FUNCTION_BLOCK FB_Homing_Base EXTENDS FB_CyclicFB IMPLEMENTS I_HomingStrategy
VAR
    _Axis     : SPT_Motion_Control.I_BasicAxis;
    _bBusy    : BOOL;
    _bDone    : BOOL;
    _bError   : BOOL;
    _bErrorID : UDINT;
    nStep     : INT;
END_VAR

METHOD Abort
VAR_INPUT
END_VAR
_bBusy := FALSE;
nStep := 0;
END_METHOD

PROPERTY Axis : SPT_Motion_Control.I_BasicAxis
GET
Axis := _Axis;
END_GET
SET
_Axis := Axis;
END_SET
END_PROPERTY

PROPERTY Busy : BOOL
GET
Busy := _bBusy;
END_GET
END_PROPERTY

METHOD CyclicLogic
// Pusta metoda w klasie bazowej - musi być nadpisana przez dzieci!
END_METHOD

PROPERTY Done : BOOL
GET
Done := _bDone;
END_GET
END_PROPERTY

PROPERTY Error : BOOL
GET
Error := _bError;
END_GET
END_PROPERTY

PROPERTY ErrorID : UDINT
GET
ErrorID := _bErrorID;
END_GET
END_PROPERTY

METHOD Execute : BOOL
IF _Axis = 0 THEN RETURN; END_IF

_bBusy       := TRUE;
_bDone       := FALSE;
_bError      := FALSE;
_bErrorID    := 0;
nStep        := 10; // Start sekwencji
Execute      := TRUE;
END_METHOD

PROPERTY InitComplete : BOOL
GET
InitComplete := TRUE;
END_GET
END_PROPERTY

END_FUNCTION_BLOCK

(* stored: Version 1.1.0.1, ProductVersion 3.1.4024.15
   POU FB_Homing_Base: Id {096ab850-5bfb-43e7-92b1-cebcdc4c0545}, SpecialFunc None
   Method Abort: Id {11111111-1111-4444-aaaa-111111111111}
   Property Axis: Id {22222222-2222-4444-aaaa-222222222222}
   Get Get: Id {33333333-3333-4444-aaaa-333333333333}
   Set Set: Id {44444444-4444-4444-aaaa-444444444444}
   Property Busy: Id {55555555-5555-4444-aaaa-555555555555}
   Get Get: Id {66666666-6666-4444-aaaa-666666666666}
   Method CyclicLogic: Id {77777777-7777-4444-aaaa-777777777777}
   Property Done: Id {88888888-8888-4444-aaaa-888888888888}
   Get Get: Id {99999999-9999-4444-aaaa-999999999999}
   Property Error: Id {aaaaaaaa-aaaa-4444-aaaa-aaaaaaaaaaaa}
   Get Get: Id {bbbbbbbb-bbbb-4444-aaaa-bbbbbbbbbbbb}
   Property ErrorID: Id {cccccccc-cccc-4444-aaaa-cccccccccccc}
   Get Get: Id {dddddddd-dddd-4444-aaaa-dddddddddddd}
   Method Execute: Id {eeeeeeee-eeee-4444-aaaa-eeeeeeeeeeee}
   Property InitComplete: Id {ffffffff-ffff-4444-aaaa-ffffffffffff}
   Get Get: Id {00000000-0000-5555-bbbb-000000000000} *)
